{attribute 'Tc2GvlVarNames'}
VAR_GLOBAL RETAIN

END_VAR

(* stored: Version 1.1.0.1, ProductVersion 3.1.4024.9
   GVL Setup_Data: Id {fc8185bd-7aeb-4e3c-9783-803a9070c079} *)
